// TIA Portal V18 export
FUNCTION "Block_2" : Void   // FC2, LAD
{ S7_Optimized_Access := 'TRUE' }
VERSION : 0.1
// stored: AutoNumber true, IsIECCheckEnabled false, SetENOAutomatically false, UDAEnableTagReadback false
   VAR_INPUT
      test : Int;
   END_VAR
   VAR_OUTPUT
      test_out : Bool;
   END_VAR
BEGIN

REGION Network 1
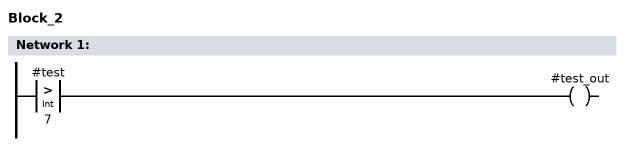
   RUNG wire#powerrail
      { S7_Templates := "SrcType := Int" } GT_Contact(in1 := #test, in2 := 7)
      Coil( #test_out )
   END_RUNG
   // the same network as SCL:
   #test_out := #test > 7;
END_REGION
END_FUNCTION
